KUKA KRL data list: MatLabControl.dat

&ACCESS RVP
&REL 4
DEFDAT  MATLABCONTROL PUBLIC

DECL GLOBAL POS target_pos={X 509.876,Y 339.917,Z 552.366,A 0.0,B 90.0000,C 0.0} ; Default safe position
DECL GLOBAL BOOL move_trigger=TRUE ; Flag to trigger movement

ENDDAT
